FUNCTION_BLOCK DecoratorBase IMPLEMENTS ITF_Analogue
VAR
	wrappee : ITF_Analogue;
END_VAR

METHOD GetValue : LREAL
END_METHOD

PROPERTY MyWrappee : itf_analogue
GET
MyWrappee := wrappee;
END_GET
SET
wrappee := MyWrappee;
END_SET
END_PROPERTY

END_FUNCTION_BLOCK

(* stored: Version 1.1.0.1, ProductVersion 3.1.4024.12
   POU DecoratorBase: Id {1cb74713-3c8c-45d1-a0fd-959659e4b46f}, SpecialFunc None
   Method GetValue: Id {d204e14d-39c6-4f66-8b66-04a44c2c3614}
   Property MyWrappee: Id {eb7cabae-0d06-4c6a-99e0-5bc98b30dd14}
   Get Get: Id {82e649fd-4cf8-473e-bac5-0670e47f5f7b}
   Set Set: Id {22b53e0c-d5d2-404f-92d2-92f8187c3bb1} *)
